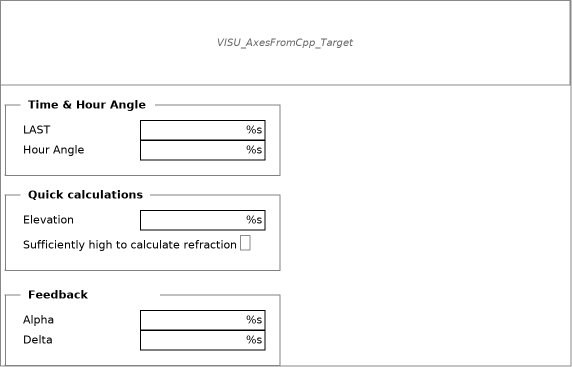
VISUALIZATION VISU_AxesFromCpp  // 572x367
VAR_IN_OUT
	ref : Axes;
    widget : AxesWidget;
END_VAR
    Polyline (20,105) (5,105) (5,175) (280,175) (280,105) (155,105)
    Label (20,120 80x20), "LAST"
    Rectangle (140,120 125x20), "%s", text variable: widget.last.hmsString
    Label (25,95 125x20), "Time & Hour Angle"
    Polyline (20,295) (5,295) (5,365) (280,365) (280,295) (160,295)
    Label (25,285 130x20), "Feedback"
    Label (20,310 105x20), "Alpha"
    Label (20,330 80x20), "Delta"
    Rectangle (140,310 125x20), "%s", text variable: widget.feedback.alpha.hmsString
    Rectangle (140,330 125x20), "%s", text variable: widget.feedback.delta.dmsString
    Label (20,140 80x20), "Hour Angle"
    Rectangle (140,140 125x20), "%s", text variable: widget.ha.hmsString
    Polyline (20,195) (5,195) (5,270) (280,270) (280,195) (150,195)
    Label (25,185 130x20), "Quick calculations"
    Label (20,210 105x20), "Elevation"
    Rectangle (140,210 125x20), "%s", text variable: widget.quickElevation.dmsString
    Frame (0,0 570x85)
        shows VISU_AxesFromCpp_Target(ref := ref, widget := widget)
    Label (20,235 225x20), "Sufficiently high to calculate refraction"
    Frame (240,235 10x15)
        shows VISU_State_green_red(state := ref.target.isTooLow)
END_VISUALIZATION

(* stored: Version 1.1.0.1, ProductVersion 3.1.4019.2
   Visu VISU_AxesFromCpp: Id {40c8445f-5d90-437c-ac04-8b82b687eb6e} *)
